ABB RAPID module: Module1.mod

MODULE Module1

! ## =========================================================================== ##
    ! MIT License
    ! Copyright (c) 2021 Roman Parak
    ! Permission is hereby granted, free of charge, to any person obtaining a copy
    ! of this software and associated documentation files (the "Software"), to deal
    ! in the Software without restriction, including without limitation the rights
    ! to use, copy, modify, merge, publish, distribute, sublicense, and/or sell
    ! copies of the Software, and to permit persons to whom the Software is
    ! furnished to do so, subject to the following conditions:
    ! The above copyright notice and this permission notice shall be included in all
    ! copies or substantial portions of the Software.
    ! THE SOFTWARE IS PROVIDED "AS IS", WITHOUT WARRANTY OF ANY KIND, EXPRESS OR
    ! IMPLIED, INCLUDING BUT NOT LIMITED TO THE WARRANTIES OF MERCHANTABILITY,
    ! FITNESS FOR A PARTICULAR PURPOSE AND NONINFRINGEMENT. IN NO EVENT SHALL THE
    ! AUTHORS OR COPYRIGHT HOLDERS BE LIABLE FOR ANY CLAIM, DAMAGES OR OTHER
    ! LIABILITY, WHETHER IN AN ACTION OF CONTRACT, TORT OR OTHERWISE, ARISING FROM,
    ! OUT OF OR IN CONNECTION WITH THE SOFTWARE OR THE USE OR OTHER DEALINGS IN THE
    ! SOFTWARE.
    ! ## =========================================================================== ##
    ! Author   : Roman Parak
    ! Email    : Roman.Parak@outlook.com
    ! Github   : https://github.com/rparak
    ! File Name: T_ROB1/Module1.mod
    ! ## =========================================================================== ##

    ! ############### EGM Initialization Parameters ############### !
    ! Identifier for the EGM correction.
     VAR robtarget starting_position;

    ! ################################## Externally Guided motion (EGM) - Main Cycle ################################## !
    PROC main()
        starting_position := CRobT(\Tool:=Tooldata_7\wobj:=wobj0);
        MoveJ RelTool (starting_position, 327, 6, -563 \Rx:=-9.8, \Ry:=17.7, \Rz:=0), v400, z1, Tooldata_7;
        MoveJ RelTool (starting_position, 326, 8, -564 \Rx:=-9.9, \Ry:=17.4, \Rz:=0), v400, z1, Tooldata_7;
        MoveJ RelTool (starting_position, 325, 10, -565 \Rx:=-9.9, \Ry:=17.1, \Rz:=0), v400, z1, Tooldata_7;
        MoveJ RelTool (starting_position, 324, 12, -566 \Rx:=-9.9, \Ry:=17.1, \Rz:=0), v400, z1, Tooldata_7;
        MoveJ RelTool (starting_position, 323, 14, -567 \Rx:=-9.9, \Ry:=16.8, \Rz:=0), v400, z1, Tooldata_7;
        MoveJ RelTool (starting_position, 321, 16, -568 \Rx:=-9.9, \Ry:=16.5, \Rz:=0), v400, z1, Tooldata_7;
        MoveJ RelTool (starting_position, 320, 20, -569 \Rx:=-10, \Ry:=16.2, \Rz:=0), v400, z1, Tooldata_7;
        MoveJ RelTool (starting_position, 318, 22, -570 \Rx:=-10, \Ry:=15.9, \Rz:=0), v400, z1, Tooldata_7;
        MoveJ RelTool (starting_position, 317, 26, -571 \Rx:=-10, \Ry:=15.6, \Rz:=0), v400, z1, Tooldata_7;
        MoveJ RelTool (starting_position, 315, 28, -572 \Rx:=-10, \Ry:=15.6, \Rz:=0), v400, z1, Tooldata_7;
        MoveJ RelTool (starting_position, 313, 32, -573 \Rx:=-10, \Ry:=15.3, \Rz:=0), v400, z1, Tooldata_7;
        MoveJ RelTool (starting_position, 311, 34, -574 \Rx:=-10, \Ry:=15, \Rz:=0), v400, z1, Tooldata_7;
        MoveJ RelTool (starting_position, 309, 38, -576 \Rx:=-10, \Ry:=14.7, \Rz:=0), v400, z1, Tooldata_7;
        MoveJ RelTool (starting_position, 307, 42, -577 \Rx:=-10, \Ry:=14.4, \Rz:=0), v400, z1, Tooldata_7;
        MoveJ RelTool (starting_position, 305, 44, -578 \Rx:=-9.9, \Ry:=14.1, \Rz:=0), v400, z1, Tooldata_7;
        MoveJ RelTool (starting_position, 302, 48, -580 \Rx:=-9.9, \Ry:=13.8, \Rz:=0), v400, z1, Tooldata_7;
        MoveJ RelTool (starting_position, 300, 52, -581 \Rx:=-9.8, \Ry:=13.5, \Rz:=0), v400, z1, Tooldata_7;
        MoveJ RelTool (starting_position, 298, 54, -583 \Rx:=-9.8, \Ry:=13.2, \Rz:=0), v400, z1, Tooldata_7;
        MoveJ RelTool (starting_position, 296, 58, -584 \Rx:=-9.7, \Ry:=12.9, \Rz:=0), v400, z1, Tooldata_7;
        MoveJ RelTool (starting_position, 293, 62, -586 \Rx:=-9.5, \Ry:=12.6, \Rz:=0), v400, z1, Tooldata_7;
        MoveJ RelTool (starting_position, 291, 64, -587 \Rx:=-9.4, \Ry:=12.3, \Rz:=0), v400, z1, Tooldata_7;
        MoveJ RelTool (starting_position, 288, 68, -589 \Rx:=-9.3, \Ry:=12, \Rz:=0), v400, z1, Tooldata_7;
        MoveJ RelTool (starting_position, 285, 72, -590 \Rx:=-9.2, \Ry:=11.7, \Rz:=0), v400, z1, Tooldata_7;
        MoveJ RelTool (starting_position, 283, 74, -592 \Rx:=-9.2, \Ry:=11.1, \Rz:=0), v400, z1, Tooldata_7;
        MoveJ RelTool (starting_position, 280, 78, -594 \Rx:=-9.1, \Ry:=10.8, \Rz:=0), v400, z1, Tooldata_7;
        MoveJ RelTool (starting_position, 277, 82, -595 \Rx:=-8.9, \Ry:=10.5, \Rz:=0), v400, z1, Tooldata_7;
        MoveJ RelTool (starting_position, 274, 84, -597 \Rx:=-8.8, \Ry:=10.2, \Rz:=0), v400, z1, Tooldata_7;
        MoveJ RelTool (starting_position, 270, 88, -598 \Rx:=-8.7, \Ry:=9.6, \Rz:=0), v400, z1, Tooldata_7;
        MoveJ RelTool (starting_position, 267, 92, -600 \Rx:=-8.6, \Ry:=9, \Rz:=0), v400, z1, Tooldata_7;
        MoveJ RelTool (starting_position, 263, 94, -601 \Rx:=-8.5, \Ry:=8.7, \Rz:=0), v400, z1, Tooldata_7;
        MoveJ RelTool (starting_position, 260, 98, -603 \Rx:=-8.4, \Ry:=8.1, \Rz:=0), v400, z1, Tooldata_7;
        MoveJ RelTool (starting_position, 256, 102, -604 \Rx:=-8.2, \Ry:=7.5, \Rz:=0), v400, z1, Tooldata_7;
        MoveJ RelTool (starting_position, 253, 104, -605 \Rx:=-8.1, \Ry:=6.9, \Rz:=0), v400, z1, Tooldata_7;
        MoveJ RelTool (starting_position, 249, 108, -606 \Rx:=-7.9, \Ry:=6.6, \Rz:=0), v400, z1, Tooldata_7;
        MoveJ RelTool (starting_position, 245, 112, -607 \Rx:=-7.6, \Ry:=6, \Rz:=0), v400, z1, Tooldata_7;
        MoveJ RelTool (starting_position, 242, 114, -608 \Rx:=-7.4, \Ry:=5.7, \Rz:=0), v400, z1, Tooldata_7;
        MoveJ RelTool (starting_position, 238, 118, -609 \Rx:=-7.1, \Ry:=5.1, \Rz:=0), v400, z1, Tooldata_7;
        MoveJ RelTool (starting_position, 234, 122, -609 \Rx:=-6.8, \Ry:=4.5, \Rz:=0), v400, z1, Tooldata_7;
        MoveJ RelTool (starting_position, 231, 124, -610 \Rx:=-6.6, \Ry:=4.2, \Rz:=0), v400, z1, Tooldata_7;
        MoveJ RelTool (starting_position, 227, 128, -610 \Rx:=-6.4, \Ry:=3.6, \Rz:=0), v400, z1, Tooldata_7;
        MoveJ RelTool (starting_position, 224, 130, -611 \Rx:=-6.1, \Ry:=3.3, \Rz:=0), v400, z1, Tooldata_7;
        MoveJ RelTool (starting_position, 220, 134, -611 \Rx:=-6, \Ry:=2.7, \Rz:=0), v400, z1, Tooldata_7;
        MoveJ RelTool (starting_position, 217, 136, -611 \Rx:=-5.9, \Ry:=2.1, \Rz:=0), v400, z1, Tooldata_7;
        MoveJ RelTool (starting_position, 213, 140, -611 \Rx:=-5.9, \Ry:=1.5, \Rz:=0), v400, z1, Tooldata_7;
        MoveJ RelTool (starting_position, 210, 142, -611 \Rx:=-5.9, \Ry:=1.2, \Rz:=0), v400, z1, Tooldata_7;
        MoveJ RelTool (starting_position, 207, 146, -611 \Rx:=-5.9, \Ry:=0.9, \Rz:=0), v400, z1, Tooldata_7;
        MoveJ RelTool (starting_position, 203, 148, -611 \Rx:=-6, \Ry:=0.3, \Rz:=0), v400, z1, Tooldata_7;
        MoveJ RelTool (starting_position, 200, 152, -610 \Rx:=-6.2, \Ry:=0, \Rz:=0), v400, z1, Tooldata_7;
        MoveJ RelTool (starting_position, 198, 156, -610 \Rx:=-6.4, \Ry:=-0.3, \Rz:=0), v400, z1, Tooldata_7;
        MoveJ RelTool (starting_position, 195, 158, -610 \Rx:=-6.6, \Ry:=-0.9, \Rz:=0), v400, z1, Tooldata_7;
        MoveJ RelTool (starting_position, 192, 162, -609 \Rx:=-6.8, \Ry:=-1.2, \Rz:=0), v400, z1, Tooldata_7;
        MoveJ RelTool (starting_position, 190, 164, -609 \Rx:=-7.1, \Ry:=-1.5, \Rz:=0), v400, z1, Tooldata_7;
        MoveJ RelTool (starting_position, 188, 168, -608 \Rx:=-7.5, \Ry:=-1.8, \Rz:=0), v400, z1, Tooldata_7;
        MoveJ RelTool (starting_position, 186, 170, -608 \Rx:=-7.8, \Ry:=-2.1, \Rz:=0), v400, z1, Tooldata_7;
        MoveJ RelTool (starting_position, 184, 174, -607 \Rx:=-8.2, \Ry:=-2.4, \Rz:=0), v400, z1, Tooldata_7;
        MoveJ RelTool (starting_position, 182, 176, -607 \Rx:=-8.7, \Ry:=-2.7, \Rz:=0), v400, z1, Tooldata_7;
        MoveJ RelTool (starting_position, 180, 180, -607 \Rx:=-9.1, \Ry:=-2.7, \Rz:=0), v400, z1, Tooldata_7;
        MoveJ RelTool (starting_position, 179, 182, -606 \Rx:=-9.4, \Ry:=-3, \Rz:=0), v400, z1, Tooldata_7;
        MoveJ RelTool (starting_position, 178, 186, -605 \Rx:=-9.8, \Ry:=-3, \Rz:=0), v400, z1, Tooldata_7;
        MoveJ RelTool (starting_position, 177, 188, -605 \Rx:=-10.2, \Ry:=-3.3, \Rz:=0), v400, z1, Tooldata_7;
        MoveJ RelTool (starting_position, 176, 192, -604 \Rx:=-10.6, \Ry:=-3.3, \Rz:=0), v400, z1, Tooldata_7;
        MoveJ RelTool (starting_position, 175, 194, -604 \Rx:=-11, \Ry:=-3.3, \Rz:=0), v400, z1, Tooldata_7;
        MoveJ RelTool (starting_position, 174, 198, -603 \Rx:=-11.3, \Ry:=-3.6, \Rz:=0), v400, z1, Tooldata_7;
        MoveJ RelTool (starting_position, 173, 200, -603 \Rx:=-11.7, \Ry:=-3.6, \Rz:=0), v400, z1, Tooldata_7;
        MoveJ RelTool (starting_position, 173, 202, -602 \Rx:=-12.1, \Ry:=-3.6, \Rz:=0), v400, z1, Tooldata_7;
        MoveJ RelTool (starting_position, 172, 206, -601 \Rx:=-12.4, \Ry:=-3.9, \Rz:=0), v400, z1, Tooldata_7;
        MoveJ RelTool (starting_position, 172, 208, -601 \Rx:=-12.7, \Ry:=-3.9, \Rz:=0), v400, z1, Tooldata_7;
        MoveJ RelTool (starting_position, 172, 212, -600 \Rx:=-12.9, \Ry:=-3.9, \Rz:=0), v400, z1, Tooldata_7;
        MoveJ RelTool (starting_position, 172, 214, -599 \Rx:=-13, \Ry:=-3.9, \Rz:=0), v400, z1, Tooldata_7;
        MoveJ RelTool (starting_position, 172, 218, -599 \Rx:=-13.1, \Ry:=-3.9, \Rz:=0), v400, z1, Tooldata_7;
        MoveJ RelTool (starting_position, 172, 220, -598 \Rx:=-13.1, \Ry:=-3.9, \Rz:=0), v400, z1, Tooldata_7;
        MoveJ RelTool (starting_position, 172, 222, -597 \Rx:=-13, \Ry:=-3.6, \Rz:=0), v400, z1, Tooldata_7;
        MoveJ RelTool (starting_position, 173, 226, -597 \Rx:=-12.9, \Ry:=-3.6, \Rz:=0), v400, z1, Tooldata_7;
        MoveJ RelTool (starting_position, 173, 228, -596 \Rx:=-12.5, \Ry:=-3.6, \Rz:=0), v400, z1, Tooldata_7;
        MoveJ RelTool (starting_position, 173, 230, -595 \Rx:=-12.2, \Ry:=-3.6, \Rz:=0), v400, z1, Tooldata_7;
        MoveJ RelTool (starting_position, 174, 234, -595 \Rx:=-11.8, \Ry:=-3.6, \Rz:=0), v400, z1, Tooldata_7;
        MoveJ RelTool (starting_position, 174, 236, -594 \Rx:=-11.3, \Ry:=-3.3, \Rz:=0), v400, z1, Tooldata_7;
        MoveJ RelTool (starting_position, 175, 238, -594 \Rx:=-10.7, \Ry:=-3.3, \Rz:=0), v400, z1, Tooldata_7;
        MoveJ RelTool (starting_position, 175, 242, -593 \Rx:=-10, \Ry:=-3.3, \Rz:=0), v400, z1, Tooldata_7;
        MoveJ RelTool (starting_position, 175, 244, -593 \Rx:=-9.2, \Ry:=-3.3, \Rz:=0), v400, z1, Tooldata_7;
        MoveJ RelTool (starting_position, 176, 246, -592 \Rx:=-8.4, \Ry:=-3.3, \Rz:=0), v400, z1, Tooldata_7;
        MoveJ RelTool (starting_position, 176, 248, -592 \Rx:=-7.6, \Ry:=-3, \Rz:=0), v400, z1, Tooldata_7;
        MoveJ RelTool (starting_position, 176, 252, -591 \Rx:=-6.7, \Ry:=-3, \Rz:=0), v400, z1, Tooldata_7;
        MoveJ RelTool (starting_position, 177, 254, -591 \Rx:=-5.8, \Ry:=-3, \Rz:=0), v400, z1, Tooldata_7;
        MoveJ RelTool (starting_position, 177, 258, -591 \Rx:=-5, \Ry:=-3, \Rz:=0), v400, z1, Tooldata_7;
        MoveJ RelTool (starting_position, 177, 260, -591 \Rx:=-4.2, \Ry:=-3, \Rz:=0), v400, z1, Tooldata_7;
        MoveJ RelTool (starting_position, 176, 262, -590 \Rx:=-3.5, \Ry:=-3, \Rz:=0), v400, z1, Tooldata_7;
        MoveJ RelTool (starting_position, 176, 266, -590 \Rx:=-2.8, \Ry:=-3, \Rz:=0), v400, z1, Tooldata_7;
        MoveJ RelTool (starting_position, 176, 268, -590 \Rx:=-2.2, \Ry:=-3, \Rz:=0), v400, z1, Tooldata_7;
        MoveJ RelTool (starting_position, 175, 270, -590 \Rx:=-1.5, \Ry:=-3.3, \Rz:=0), v400, z1, Tooldata_7;
        MoveJ RelTool (starting_position, 174, 274, -590 \Rx:=-1, \Ry:=-3.3, \Rz:=0), v400, z1, Tooldata_7;
        MoveJ RelTool (starting_position, 173, 276, -590 \Rx:=-0.5, \Ry:=-3.3, \Rz:=0), v400, z1, Tooldata_7;
        MoveJ RelTool (starting_position, 172, 278, -590 \Rx:=-0.1, \Ry:=-3.6, \Rz:=0), v400, z1, Tooldata_7;
        MoveJ RelTool (starting_position, 170, 280, -590 \Rx:=0.2, \Ry:=-3.6, \Rz:=0), v400, z1, Tooldata_7;
        MoveJ RelTool (starting_position, 168, 282, -590 \Rx:=0.5, \Ry:=-3.9, \Rz:=0), v400, z1, Tooldata_7;
        MoveJ RelTool (starting_position, 166, 284, -590 \Rx:=0.6, \Ry:=-4.2, \Rz:=0), v400, z1, Tooldata_7;
        MoveJ RelTool (starting_position, 164, 286, -590 \Rx:=0.6, \Ry:=-4.5, \Rz:=0), v400, z1, Tooldata_7;
        MoveJ RelTool (starting_position, 161, 288, -590 \Rx:=0.6, \Ry:=-4.8, \Rz:=0), v400, z1, Tooldata_7;
        MoveJ RelTool (starting_position, 159, 292, -590 \Rx:=0.6, \Ry:=-5.4, \Rz:=0), v400, z1, Tooldata_7;
        MoveJ RelTool (starting_position, 155, 294, -590 \Rx:=0.6, \Ry:=-5.7, \Rz:=0), v400, z1, Tooldata_7;
        MoveJ RelTool (starting_position, 152, 296, -589 \Rx:=0.5, \Ry:=-6.3, \Rz:=0), v400, z1, Tooldata_7;
        MoveJ RelTool (starting_position, 149, 298, -589 \Rx:=0.4, \Ry:=-6.6, \Rz:=0), v400, z1, Tooldata_7;
        MoveJ RelTool (starting_position, 145, 300, -589 \Rx:=0.4, \Ry:=-7.2, \Rz:=0), v400, z1, Tooldata_7;
        MoveJ RelTool (starting_position, 141, 302, -588 \Rx:=0.3, \Ry:=-7.8, \Rz:=0), v400, z1, Tooldata_7;
        MoveJ RelTool (starting_position, 137, 304, -588 \Rx:=0.3, \Ry:=-8.4, \Rz:=0), v400, z1, Tooldata_7;
        MoveJ RelTool (starting_position, 133, 306, -587 \Rx:=0.4, \Ry:=-9, \Rz:=0), v400, z1, Tooldata_7;
        MoveJ RelTool (starting_position, 129, 308, -586 \Rx:=0.4, \Ry:=-9.6, \Rz:=0), v400, z1, Tooldata_7;
        MoveJ RelTool (starting_position, 125, 310, -586 \Rx:=0.5, \Ry:=-10.2, \Rz:=0), v400, z1, Tooldata_7;
        MoveJ RelTool (starting_position, 120, 314, -585 \Rx:=0.6, \Ry:=-10.5, \Rz:=0), v400, z1, Tooldata_7;
        MoveJ RelTool (starting_position, 116, 316, -583 \Rx:=0.9, \Ry:=-11.1, \Rz:=0), v400, z1, Tooldata_7;
        MoveJ RelTool (starting_position, 111, 318, -582 \Rx:=1.2, \Ry:=-11.7, \Rz:=0), v400, z1, Tooldata_7;
        MoveJ RelTool (starting_position, 107, 318, -581 \Rx:=1.5, \Ry:=-12.3, \Rz:=0), v400, z1, Tooldata_7;
        MoveJ RelTool (starting_position, 102, 320, -579 \Rx:=1.9, \Ry:=-12.9, \Rz:=0), v400, z1, Tooldata_7;
        MoveJ RelTool (starting_position, 97, 322, -577 \Rx:=2.4, \Ry:=-13.8, \Rz:=0), v400, z1, Tooldata_7;
        MoveJ RelTool (starting_position, 92, 324, -575 \Rx:=2.8, \Ry:=-14.7, \Rz:=0), v400, z1, Tooldata_7;
        MoveJ RelTool (starting_position, 88, 326, -573 \Rx:=3.2, \Ry:=-15.3, \Rz:=0), v400, z1, Tooldata_7;
        MoveJ RelTool (starting_position, 83, 328, -571 \Rx:=3.7, \Ry:=-15.9, \Rz:=0), v400, z1, Tooldata_7;
        MoveJ RelTool (starting_position, 79, 330, -569 \Rx:=4.2, \Ry:=-16.5, \Rz:=0), v400, z1, Tooldata_7;
        MoveJ RelTool (starting_position, 74, 332, -566 \Rx:=4.7, \Ry:=-17.1, \Rz:=0), v400, z1, Tooldata_7;
        MoveJ RelTool (starting_position, 70, 334, -564 \Rx:=5.2, \Ry:=-17.7, \Rz:=0), v400, z1, Tooldata_7;
        MoveJ RelTool (starting_position, 66, 336, -561 \Rx:=5.6, \Ry:=-18, \Rz:=0), v400, z1, Tooldata_7;
        MoveJ RelTool (starting_position, 62, 338, -558 \Rx:=6.2, \Ry:=-18.6, \Rz:=0), v400, z1, Tooldata_7;
        MoveJ RelTool (starting_position, 59, 340, -555 \Rx:=6.7, \Ry:=-19.2, \Rz:=0), v400, z1, Tooldata_7;
        MoveJ RelTool (starting_position, 55, 342, -553 \Rx:=7.2, \Ry:=-19.5, \Rz:=0), v400, z1, Tooldata_7;
        MoveJ RelTool (starting_position, 52, 344, -550 \Rx:=7.6, \Ry:=-20.1, \Rz:=0), v400, z1, Tooldata_7;
        MoveJ RelTool (starting_position, 49, 344, -546 \Rx:=8.1, \Ry:=-20.4, \Rz:=0), v400, z1, Tooldata_7;
        MoveJ RelTool (starting_position, 46, 346, -543 \Rx:=8.6, \Ry:=-21, \Rz:=0), v400, z1, Tooldata_7;
        MoveJ RelTool (starting_position, 44, 348, -540 \Rx:=9, \Ry:=-21.3, \Rz:=0), v400, z1, Tooldata_7;
        MoveJ RelTool (starting_position, 41, 350, -537 \Rx:=9.4, \Ry:=-21.3, \Rz:=0), v400, z1, Tooldata_7;
        MoveJ RelTool (starting_position, 39, 352, -534 \Rx:=9.8, \Ry:=-21.9, \Rz:=0), v400, z1, Tooldata_7;
        MoveJ RelTool (starting_position, 37, 354, -530 \Rx:=10.2, \Ry:=-22.2, \Rz:=0), v400, z1, Tooldata_7;
        MoveJ RelTool (starting_position, 36, 356, -527 \Rx:=10.6, \Ry:=-22.2, \Rz:=0), v400, z1, Tooldata_7;
        MoveJ RelTool (starting_position, 34, 358, -524 \Rx:=10.9, \Ry:=-22.5, \Rz:=0), v400, z1, Tooldata_7;
        MoveJ RelTool (starting_position, 33, 358, -521 \Rx:=11.2, \Ry:=-22.5, \Rz:=0), v400, z1, Tooldata_7;
        MoveJ RelTool (starting_position, 32, 360, -517 \Rx:=11.5, \Ry:=-22.8, \Rz:=0), v400, z1, Tooldata_7;
        MoveJ RelTool (starting_position, 32, 360, -514 \Rx:=11.9, \Ry:=-22.8, \Rz:=0), v400, z1, Tooldata_7;
        MoveJ RelTool (starting_position, 31, 362, -511 \Rx:=12.2, \Ry:=-22.8, \Rz:=0), v400, z1, Tooldata_7;
        MoveJ RelTool (starting_position, 31, 362, -507 \Rx:=12.5, \Ry:=-22.8, \Rz:=0), v400, z1, Tooldata_7;
        MoveJ RelTool (starting_position, 31, 364, -504 \Rx:=12.8, \Ry:=-22.8, \Rz:=0), v400, z1, Tooldata_7;
        MoveJ RelTool (starting_position, 31, 366, -501 \Rx:=13, \Ry:=-22.8, \Rz:=0), v400, z1, Tooldata_7;
        MoveJ RelTool (starting_position, 31, 366, -498 \Rx:=13.3, \Ry:=-22.8, \Rz:=0), v400, z1, Tooldata_7;
        MoveJ RelTool (starting_position, 31, 368, -495 \Rx:=13.5, \Ry:=-22.8, \Rz:=0), v400, z1, Tooldata_7;
        MoveJ RelTool (starting_position, 31, 370, -492 \Rx:=13.7, \Ry:=-22.8, \Rz:=0), v400, z1, Tooldata_7;
        MoveJ RelTool (starting_position, 32, 372, -488 \Rx:=13.9, \Ry:=-22.8, \Rz:=0), v400, z1, Tooldata_7;
        MoveJ RelTool (starting_position, 32, 374, -485 \Rx:=14.1, \Ry:=-22.5, \Rz:=0), v400, z1, Tooldata_7;
        MoveJ RelTool (starting_position, 33, 376, -482 \Rx:=14.2, \Ry:=-22.5, \Rz:=0), v400, z1, Tooldata_7;
        MoveJ RelTool (starting_position, 34, 378, -479 \Rx:=14.3, \Ry:=-22.2, \Rz:=0), v400, z1, Tooldata_7;
        MoveJ RelTool (starting_position, 35, 378, -476 \Rx:=14.3, \Ry:=-22.2, \Rz:=0), v400, z1, Tooldata_7;
        MoveJ RelTool (starting_position, 36, 380, -473 \Rx:=14.3, \Ry:=-22.2, \Rz:=0), v400, z1, Tooldata_7;
        MoveJ RelTool (starting_position, 37, 380, -470 \Rx:=14.2, \Ry:=-21.9, \Rz:=0), v400, z1, Tooldata_7;
        MoveJ RelTool (starting_position, 38, 380, -467 \Rx:=14.1, \Ry:=-21.6, \Rz:=0), v400, z1, Tooldata_7;
        MoveJ RelTool (starting_position, 39, 380, -465 \Rx:=13.8, \Ry:=-21.6, \Rz:=0), v400, z1, Tooldata_7;
        MoveJ RelTool (starting_position, 40, 380, -462 \Rx:=13.5, \Ry:=-21.3, \Rz:=0), v400, z1, Tooldata_7;
        MoveJ RelTool (starting_position, 41, 380, -459 \Rx:=13.1, \Ry:=-21.3, \Rz:=0), v400, z1, Tooldata_7;
        MoveJ RelTool (starting_position, 43, 380, -456 \Rx:=12.6, \Ry:=-21, \Rz:=0), v400, z1, Tooldata_7;
        MoveJ RelTool (starting_position, 44, 380, -453 \Rx:=12.1, \Ry:=-21, \Rz:=0), v400, z1, Tooldata_7;
        MoveJ RelTool (starting_position, 45, 382, -451 \Rx:=11.5, \Ry:=-20.7, \Rz:=0), v400, z1, Tooldata_7;
        MoveJ RelTool (starting_position, 46, 382, -448 \Rx:=10.8, \Ry:=-20.7, \Rz:=0), v400, z1, Tooldata_7;
        MoveJ RelTool (starting_position, 47, 384, -445 \Rx:=10.1, \Ry:=-20.4, \Rz:=0), v400, z1, Tooldata_7;
        MoveJ RelTool (starting_position, 48, 386, -442 \Rx:=9.2, \Ry:=-20.4, \Rz:=0), v400, z1, Tooldata_7;
        MoveJ RelTool (starting_position, 49, 386, -440 \Rx:=8.3, \Ry:=-20.1, \Rz:=0), v400, z1, Tooldata_7;
        MoveJ RelTool (starting_position, 50, 388, -437 \Rx:=7.3, \Ry:=-20.1, \Rz:=0), v400, z1, Tooldata_7;
        MoveJ RelTool (starting_position, 51, 390, -434 \Rx:=6.3, \Ry:=-20.1, \Rz:=0), v400, z1, Tooldata_7;
        MoveJ RelTool (starting_position, 52, 392, -432 \Rx:=5.2, \Ry:=-19.8, \Rz:=0), v400, z1, Tooldata_7;
        MoveJ RelTool (starting_position, 52, 394, -429 \Rx:=4.2, \Ry:=-19.8, \Rz:=0), v400, z1, Tooldata_7;
        MoveJ RelTool (starting_position, 53, 396, -427 \Rx:=3.1, \Ry:=-19.5, \Rz:=0), v400, z1, Tooldata_7;
        MoveJ RelTool (starting_position, 54, 398, -424 \Rx:=2.1, \Ry:=-19.5, \Rz:=0), v400, z1, Tooldata_7;
        MoveJ RelTool (starting_position, 55, 398, -422 \Rx:=1.1, \Ry:=-19.5, \Rz:=0), v400, z1, Tooldata_7;
        MoveJ RelTool (starting_position, 55, 400, -419 \Rx:=0.1, \Ry:=-19.2, \Rz:=0), v400, z1, Tooldata_7;
        MoveJ RelTool (starting_position, 56, 400, -417 \Rx:=-0.9, \Ry:=-19.2, \Rz:=0), v400, z1, Tooldata_7;
        MoveJ RelTool (starting_position, 57, 400, -415 \Rx:=-1.8, \Ry:=-19.2, \Rz:=0), v400, z1, Tooldata_7;
        MoveJ RelTool (starting_position, 57, 400, -413 \Rx:=-2.6, \Ry:=-19.2, \Rz:=0), v400, z1, Tooldata_7;
        MoveJ RelTool (starting_position, 58, 400, -410 \Rx:=-3.3, \Ry:=-19.2, \Rz:=0), v400, z1, Tooldata_7;
        MoveJ RelTool (starting_position, 58, 400, -408 \Rx:=-3.8, \Ry:=-18.9, \Rz:=0), v400, z1, Tooldata_7;
        MoveJ RelTool (starting_position, 59, 400, -406 \Rx:=-4.1, \Ry:=-18.9, \Rz:=0), v400, z1, Tooldata_7;
        MoveJ RelTool (starting_position, 59, 400, -404 \Rx:=-4.4, \Ry:=-18.9, \Rz:=0), v400, z1, Tooldata_7;
        MoveJ RelTool (starting_position, 60, 400, -402 \Rx:=-4.6, \Ry:=-18.9, \Rz:=0), v400, z1, Tooldata_7;
        MoveJ RelTool (starting_position, 60, 400, -400 \Rx:=-4.6, \Ry:=-18.6, \Rz:=0), v400, z1, Tooldata_7;
        MoveJ RelTool (starting_position, 61, 400, -398 \Rx:=-4.5, \Ry:=-18.6, \Rz:=0), v400, z1, Tooldata_7;
        MoveJ RelTool (starting_position, 61, 400, -395 \Rx:=-4.2, \Ry:=-18.6, \Rz:=0), v400, z1, Tooldata_7;
        MoveJ RelTool (starting_position, 62, 400, -393 \Rx:=-3.9, \Ry:=-18.6, \Rz:=0), v400, z1, Tooldata_7;
        MoveJ RelTool (starting_position, 62, 400, -391 \Rx:=-3.4, \Ry:=-18.6, \Rz:=0), v400, z1, Tooldata_7;
        MoveJ RelTool (starting_position, 63, 400, -389 \Rx:=-2.7, \Ry:=-18.6, \Rz:=0), v400, z1, Tooldata_7;
        MoveJ RelTool (starting_position, 63, 400, -386 \Rx:=-2, \Ry:=-18.3, \Rz:=0), v400, z1, Tooldata_7;
        MoveJ RelTool (starting_position, 64, 400, -384 \Rx:=-1.3, \Ry:=-18.3, \Rz:=0), v400, z1, Tooldata_7;
        MoveJ RelTool (starting_position, 65, 400, -381 \Rx:=-0.5, \Ry:=-18.3, \Rz:=0), v400, z1, Tooldata_7;
        MoveJ RelTool (starting_position, 66, 400, -379 \Rx:=0.3, \Ry:=-18, \Rz:=0), v400, z1, Tooldata_7;
        MoveJ RelTool (starting_position, 67, 400, -376 \Rx:=1.2, \Ry:=-18, \Rz:=0), v400, z1, Tooldata_7;
        MoveJ RelTool (starting_position, 68, 400, -374 \Rx:=2, \Ry:=-17.7, \Rz:=0), v400, z1, Tooldata_7;
        MoveJ RelTool (starting_position, 70, 400, -371 \Rx:=2.9, \Ry:=-17.7, \Rz:=0), v400, z1, Tooldata_7;
        MoveJ RelTool (starting_position, 71, 400, -368 \Rx:=3.7, \Ry:=-17.4, \Rz:=0), v400, z1, Tooldata_7;
        MoveJ RelTool (starting_position, 73, 400, -366 \Rx:=4.5, \Ry:=-17.1, \Rz:=0), v400, z1, Tooldata_7;
        MoveJ RelTool (starting_position, 75, 400, -363 \Rx:=5.4, \Ry:=-17.1, \Rz:=0), v400, z1, Tooldata_7;
        MoveJ RelTool (starting_position, 77, 400, -360 \Rx:=6.2, \Ry:=-16.8, \Rz:=0), v400, z1, Tooldata_7;
        MoveJ RelTool (starting_position, 79, 400, -357 \Rx:=6.9, \Ry:=-16.2, \Rz:=0), v400, z1, Tooldata_7;
        MoveJ RelTool (starting_position, 81, 400, -355 \Rx:=7.6, \Ry:=-15.9, \Rz:=0), v400, z1, Tooldata_7;
        MoveJ RelTool (starting_position, 84, 400, -352 \Rx:=8.2, \Ry:=-15.6, \Rz:=0), v400, z1, Tooldata_7;
        MoveJ RelTool (starting_position, 86, 400, -349 \Rx:=8.8, \Ry:=-15.3, \Rz:=0), v400, z1, Tooldata_7;
        MoveJ RelTool (starting_position, 89, 400, -347 \Rx:=9.3, \Ry:=-15, \Rz:=0), v400, z1, Tooldata_7;
        MoveJ RelTool (starting_position, 92, 400, -345 \Rx:=9.7, \Ry:=-14.7, \Rz:=0), v400, z1, Tooldata_7;
        MoveJ RelTool (starting_position, 95, 400, -342 \Rx:=10.1, \Ry:=-14.1, \Rz:=0), v400, z1, Tooldata_7;
        MoveJ RelTool (starting_position, 98, 400, -340 \Rx:=10.4, \Ry:=-13.8, \Rz:=0), v400, z1, Tooldata_7;
        MoveJ RelTool (starting_position, 101, 400, -338 \Rx:=10.5, \Ry:=-13.2, \Rz:=0), v400, z1, Tooldata_7;
        MoveJ RelTool (starting_position, 104, 400, -336 \Rx:=10.6, \Ry:=-12.9, \Rz:=0), v400, z1, Tooldata_7;
        MoveJ RelTool (starting_position, 107, 400, -335 \Rx:=10.7, \Ry:=-12.3, \Rz:=0), v400, z1, Tooldata_7;
        MoveJ RelTool (starting_position, 110, 400, -333 \Rx:=10.6, \Ry:=-12, \Rz:=0), v400, z1, Tooldata_7;
        MoveJ RelTool (starting_position, 112, 400, -332 \Rx:=10.5, \Ry:=-11.7, \Rz:=0), v400, z1, Tooldata_7;
        MoveJ RelTool (starting_position, 115, 400, -331 \Rx:=10.3, \Ry:=-11.1, \Rz:=0), v400, z1, Tooldata_7;
        MoveJ RelTool (starting_position, 118, 400, -329 \Rx:=10.1, \Ry:=-10.8, \Rz:=0), v400, z1, Tooldata_7;
        MoveJ RelTool (starting_position, 120, 400, -329 \Rx:=9.9, \Ry:=-10.5, \Rz:=0), v400, z1, Tooldata_7;
        MoveJ RelTool (starting_position, 122, 398, -328 \Rx:=9.6, \Ry:=-10.2, \Rz:=0), v400, z1, Tooldata_7;
        MoveJ RelTool (starting_position, 124, 398, -327 \Rx:=9.3, \Ry:=-9.9, \Rz:=0), v400, z1, Tooldata_7;
        MoveJ RelTool (starting_position, 125, 396, -327 \Rx:=8.9, \Ry:=-9.6, \Rz:=0), v400, z1, Tooldata_7;
        MoveJ RelTool (starting_position, 127, 394, -326 \Rx:=8.6, \Ry:=-9.6, \Rz:=0), v400, z1, Tooldata_7;
        MoveJ RelTool (starting_position, 128, 394, -326 \Rx:=8.3, \Ry:=-9.3, \Rz:=0), v400, z1, Tooldata_7;
        MoveJ RelTool (starting_position, 128, 392, -325 \Rx:=8, \Ry:=-9.3, \Rz:=0), v400, z1, Tooldata_7;
        MoveJ RelTool (starting_position, 129, 390, -325 \Rx:=7.7, \Ry:=-9.3, \Rz:=0), v400, z1, Tooldata_7;
        MoveJ RelTool (starting_position, 129, 388, -325 \Rx:=7.5, \Ry:=-9.3, \Rz:=0), v400, z1, Tooldata_7;
        MoveJ RelTool (starting_position, 129, 386, -324 \Rx:=7.4, \Ry:=-9.3, \Rz:=0), v400, z1, Tooldata_7;
        MoveJ RelTool (starting_position, 128, 384, -324 \Rx:=7.3, \Ry:=-9.3, \Rz:=0), v400, z1, Tooldata_7;
        MoveJ RelTool (starting_position, 128, 382, -324 \Rx:=7.3, \Ry:=-9.3, \Rz:=0), v400, z1, Tooldata_7;
        MoveJ RelTool (starting_position, 127, 382, -323 \Rx:=7.3, \Ry:=-9.6, \Rz:=0), v400, z1, Tooldata_7;
        MoveJ RelTool (starting_position, 125, 380, -323 \Rx:=7.3, \Ry:=-9.6, \Rz:=0), v400, z1, Tooldata_7;
        MoveJ RelTool (starting_position, 124, 380, -322 \Rx:=7.4, \Ry:=-9.9, \Rz:=0), v400, z1, Tooldata_7;
        MoveJ RelTool (starting_position, 122, 380, -321 \Rx:=7.6, \Ry:=-10.2, \Rz:=0), v400, z1, Tooldata_7;
        MoveJ RelTool (starting_position, 120, 380, -321 \Rx:=7.8, \Ry:=-10.5, \Rz:=0), v400, z1, Tooldata_7;
        MoveJ RelTool (starting_position, 118, 380, -320 \Rx:=8.1, \Ry:=-10.8, \Rz:=0), v400, z1, Tooldata_7;
        MoveJ RelTool (starting_position, 115, 380, -319 \Rx:=8.3, \Ry:=-11.1, \Rz:=0), v400, z1, Tooldata_7;
        MoveJ RelTool (starting_position, 113, 380, -317 \Rx:=8.6, \Ry:=-11.7, \Rz:=0), v400, z1, Tooldata_7;
        MoveJ RelTool (starting_position, 110, 380, -316 \Rx:=8.8, \Ry:=-12, \Rz:=0), v400, z1, Tooldata_7;
        MoveJ RelTool (starting_position, 108, 378, -315 \Rx:=9.1, \Ry:=-12.6, \Rz:=0), v400, z1, Tooldata_7;
        MoveJ RelTool (starting_position, 105, 378, -313 \Rx:=9.4, \Ry:=-12.9, \Rz:=0), v400, z1, Tooldata_7;
        MoveJ RelTool (starting_position, 102, 376, -311 \Rx:=9.7, \Ry:=-13.2, \Rz:=0), v400, z1, Tooldata_7;
        MoveJ RelTool (starting_position, 100, 374, -309 \Rx:=9.9, \Ry:=-13.5, \Rz:=0), v400, z1, Tooldata_7;
        MoveJ RelTool (starting_position, 98, 374, -307 \Rx:=10.1, \Ry:=-13.8, \Rz:=0), v400, z1, Tooldata_7;
        MoveJ RelTool (starting_position, 95, 372, -305 \Rx:=10.4, \Ry:=-14.1, \Rz:=0), v400, z1, Tooldata_7;
        MoveJ RelTool (starting_position, 93, 370, -303 \Rx:=10.6, \Ry:=-14.4, \Rz:=0), v400, z1, Tooldata_7;
        MoveJ RelTool (starting_position, 91, 368, -301 \Rx:=10.7, \Ry:=-14.7, \Rz:=0), v400, z1, Tooldata_7;
        MoveJ RelTool (starting_position, 89, 366, -298 \Rx:=10.9, \Ry:=-15, \Rz:=0), v400, z1, Tooldata_7;
        MoveJ RelTool (starting_position, 88, 364, -296 \Rx:=11, \Ry:=-15.3, \Rz:=0), v400, z1, Tooldata_7;
        MoveJ RelTool (starting_position, 86, 362, -293 \Rx:=11, \Ry:=-15.6, \Rz:=0), v400, z1, Tooldata_7;
        MoveJ RelTool (starting_position, 85, 362, -291 \Rx:=11, \Ry:=-15.6, \Rz:=0), v400, z1, Tooldata_7;
        MoveJ RelTool (starting_position, 84, 360, -288 \Rx:=10.9, \Ry:=-15.9, \Rz:=0), v400, z1, Tooldata_7;
        MoveJ RelTool (starting_position, 83, 360, -286 \Rx:=10.9, \Ry:=-15.9, \Rz:=0), v400, z1, Tooldata_7;
        MoveJ RelTool (starting_position, 83, 358, -283 \Rx:=10.8, \Ry:=-16.2, \Rz:=0), v400, z1, Tooldata_7;
        MoveJ RelTool (starting_position, 82, 358, -281 \Rx:=10.7, \Ry:=-15.9, \Rz:=0), v400, z1, Tooldata_7;
        MoveJ RelTool (starting_position, 82, 356, -278 \Rx:=10.6, \Ry:=-15.9, \Rz:=0), v400, z1, Tooldata_7;
        MoveJ RelTool (starting_position, 82, 354, -275 \Rx:=10.5, \Ry:=-15.9, \Rz:=0), v400, z1, Tooldata_7;
        MoveJ RelTool (starting_position, 83, 354, -273 \Rx:=10.3, \Ry:=-15.9, \Rz:=0), v400, z1, Tooldata_7;
        MoveJ RelTool (starting_position, 83, 352, -270 \Rx:=10.2, \Ry:=-15.9, \Rz:=0), v400, z1, Tooldata_7;
        MoveJ RelTool (starting_position, 84, 350, -268 \Rx:=10.1, \Ry:=-15.6, \Rz:=0), v400, z1, Tooldata_7;
        MoveJ RelTool (starting_position, 85, 348, -266 \Rx:=9.9, \Ry:=-15.6, \Rz:=0), v400, z1, Tooldata_7;
        MoveJ RelTool (starting_position, 86, 346, -263 \Rx:=9.8, \Ry:=-15.3, \Rz:=0), v400, z1, Tooldata_7;
        MoveJ RelTool (starting_position, 88, 344, -261 \Rx:=9.7, \Ry:=-15.3, \Rz:=0), v400, z1, Tooldata_7;
        MoveJ RelTool (starting_position, 89, 342, -259 \Rx:=9.6, \Ry:=-15, \Rz:=0), v400, z1, Tooldata_7;
        MoveJ RelTool (starting_position, 90, 340, -256 \Rx:=9.5, \Ry:=-14.7, \Rz:=0), v400, z1, Tooldata_7;
        MoveJ RelTool (starting_position, 92, 338, -254 \Rx:=9.4, \Ry:=-14.4, \Rz:=0), v400, z1, Tooldata_7;
        MoveJ RelTool (starting_position, 94, 336, -252 \Rx:=9.3, \Ry:=-14.4, \Rz:=0), v400, z1, Tooldata_7;
        MoveJ RelTool (starting_position, 95, 336, -250 \Rx:=9.2, \Ry:=-14.1, \Rz:=0), v400, z1, Tooldata_7;
        MoveJ RelTool (starting_position, 97, 334, -248 \Rx:=9.2, \Ry:=-13.8, \Rz:=0), v400, z1, Tooldata_7;
        MoveJ RelTool (starting_position, 99, 332, -246 \Rx:=9.1, \Ry:=-13.5, \Rz:=0), v400, z1, Tooldata_7;
        MoveJ RelTool (starting_position, 100, 330, -245 \Rx:=9, \Ry:=-13.2, \Rz:=0), v400, z1, Tooldata_7;
        MoveJ RelTool (starting_position, 102, 326, -243 \Rx:=8.9, \Ry:=-12.9, \Rz:=0), v400, z1, Tooldata_7;
        MoveJ RelTool (starting_position, 103, 324, -241 \Rx:=8.8, \Ry:=-12.9, \Rz:=0), v400, z1, Tooldata_7;
        MoveJ RelTool (starting_position, 105, 322, -240 \Rx:=8.6, \Ry:=-12.6, \Rz:=0), v400, z1, Tooldata_7;
        MoveJ RelTool (starting_position, 106, 322, -238 \Rx:=8.5, \Ry:=-12.3, \Rz:=0), v400, z1, Tooldata_7;
        MoveJ RelTool (starting_position, 107, 320, -237 \Rx:=8.4, \Ry:=-12.3, \Rz:=0), v400, z1, Tooldata_7;
        MoveJ RelTool (starting_position, 107, 318, -236 \Rx:=8.2, \Ry:=-12.3, \Rz:=0), v400, z1, Tooldata_7;
        MoveJ RelTool (starting_position, 108, 316, -234 \Rx:=8, \Ry:=-12, \Rz:=0), v400, z1, Tooldata_7;
        MoveJ RelTool (starting_position, 108, 314, -233 \Rx:=7.8, \Ry:=-12, \Rz:=0), v400, z1, Tooldata_7;
        MoveJ RelTool (starting_position, 108, 312, -232 \Rx:=7.5, \Ry:=-12, \Rz:=0), v400, z1, Tooldata_7;
        MoveJ RelTool (starting_position, 107, 308, -232 \Rx:=7.2, \Ry:=-12, \Rz:=0), v400, z1, Tooldata_7;
        MoveJ RelTool (starting_position, 106, 306, -231 \Rx:=6.9, \Ry:=-12, \Rz:=0), v400, z1, Tooldata_7;
        MoveJ RelTool (starting_position, 105, 304, -230 \Rx:=6.6, \Ry:=-12.3, \Rz:=0), v400, z1, Tooldata_7;
        MoveJ RelTool (starting_position, 103, 302, -230 \Rx:=6.4, \Ry:=-12.6, \Rz:=0), v400, z1, Tooldata_7;
        MoveJ RelTool (starting_position, 101, 300, -229 \Rx:=6.1, \Ry:=-12.9, \Rz:=0), v400, z1, Tooldata_7;
        MoveJ RelTool (starting_position, 98, 298, -228 \Rx:=5.9, \Ry:=-13.2, \Rz:=0), v400, z1, Tooldata_7;
        MoveJ RelTool (starting_position, 95, 296, -228 \Rx:=5.7, \Ry:=-13.8, \Rz:=0), v400, z1, Tooldata_7;
        MoveJ RelTool (starting_position, 91, 294, -227 \Rx:=5.6, \Ry:=-14.1, \Rz:=0), v400, z1, Tooldata_7;
        MoveJ RelTool (starting_position, 87, 292, -227 \Rx:=5.4, \Ry:=-14.7, \Rz:=0), v400, z1, Tooldata_7;
        MoveJ RelTool (starting_position, 83, 288, -226 \Rx:=5.3, \Ry:=-15.3, \Rz:=0), v400, z1, Tooldata_7;
        MoveJ RelTool (starting_position, 79, 286, -225 \Rx:=5.3, \Ry:=-16.2, \Rz:=0), v400, z1, Tooldata_7;
        MoveJ RelTool (starting_position, 74, 284, -224 \Rx:=5.3, \Ry:=-16.8, \Rz:=0), v400, z1, Tooldata_7;
        MoveJ RelTool (starting_position, 68, 282, -223 \Rx:=5.3, \Ry:=-17.4, \Rz:=0), v400, z1, Tooldata_7;
        MoveJ RelTool (starting_position, 63, 280, -222 \Rx:=5.3, \Ry:=-18, \Rz:=0), v400, z1, Tooldata_7;
        MoveJ RelTool (starting_position, 57, 278, -220 \Rx:=5.4, \Ry:=-18.9, \Rz:=0), v400, z1, Tooldata_7;
        MoveJ RelTool (starting_position, 51, 276, -219 \Rx:=5.4, \Ry:=-19.5, \Rz:=0), v400, z1, Tooldata_7;
        MoveJ RelTool (starting_position, 45, 274, -217 \Rx:=5.5, \Ry:=-20.7, \Rz:=0), v400, z1, Tooldata_7;
        MoveJ RelTool (starting_position, 39, 270, -214 \Rx:=5.6, \Ry:=-21.6, \Rz:=0), v400, z1, Tooldata_7;
        MoveJ RelTool (starting_position, 32, 268, -212 \Rx:=5.6, \Ry:=-22.5, \Rz:=0), v400, z1, Tooldata_7;
        MoveJ RelTool (starting_position, 26, 266, -209 \Rx:=5.7, \Ry:=-23.4, \Rz:=0), v400, z1, Tooldata_7;
        MoveJ RelTool (starting_position, 19, 262, -206 \Rx:=5.8, \Ry:=-24.3, \Rz:=0), v400, z1, Tooldata_7;
        MoveJ RelTool (starting_position, 13, 260, -202 \Rx:=6, \Ry:=-25.2, \Rz:=0), v400, z1, Tooldata_7;
        MoveJ RelTool (starting_position, 6, 258, -199 \Rx:=6, \Ry:=-26.1, \Rz:=0), v400, z1, Tooldata_7;
        MoveJ RelTool (starting_position, 0, 254, -195 \Rx:=6, \Ry:=-27, \Rz:=0), v400, z1, Tooldata_7;
        MoveJ RelTool (starting_position, -6, 252, -191 \Rx:=6, \Ry:=-27.9, \Rz:=0), v400, z1, Tooldata_7;
        MoveJ RelTool (starting_position, -12, 250, -186 \Rx:=5.9, \Ry:=-28.8, \Rz:=0), v400, z1, Tooldata_7;
        MoveJ RelTool (starting_position, -18, 246, -182 \Rx:=5.8, \Ry:=-29.7, \Rz:=0), v400, z1, Tooldata_7;
        MoveJ RelTool (starting_position, -23, 244, -177 \Rx:=5.7, \Ry:=-30.3, \Rz:=0), v400, z1, Tooldata_7;
        MoveJ RelTool (starting_position, -28, 242, -172 \Rx:=5.6, \Ry:=-31.2, \Rz:=0), v400, z1, Tooldata_7;
        MoveJ RelTool (starting_position, -32, 238, -167 \Rx:=5.4, \Ry:=-31.5, \Rz:=0), v400, z1, Tooldata_7;
        MoveJ RelTool (starting_position, -36, 236, -162 \Rx:=5.2, \Ry:=-32.1, \Rz:=0), v400, z1, Tooldata_7;
        MoveJ RelTool (starting_position, -40, 234, -157 \Rx:=5, \Ry:=-32.7, \Rz:=0), v400, z1, Tooldata_7;
        MoveJ RelTool (starting_position, -43, 232, -152 \Rx:=4.7, \Ry:=-33, \Rz:=0), v400, z1, Tooldata_7;
        MoveJ RelTool (starting_position, -46, 228, -146 \Rx:=4.4, \Ry:=-33.3, \Rz:=0), v400, z1, Tooldata_7;
        MoveJ RelTool (starting_position, -48, 226, -141 \Rx:=4, \Ry:=-33.6, \Rz:=0), v400, z1, Tooldata_7;
        MoveJ RelTool (starting_position, -50, 222, -136 \Rx:=3.7, \Ry:=-33.9, \Rz:=0), v400, z1, Tooldata_7;
        MoveJ RelTool (starting_position, -51, 220, -131 \Rx:=3.4, \Ry:=-34.2, \Rz:=0), v400, z1, Tooldata_7;
        MoveJ RelTool (starting_position, -52, 218, -126 \Rx:=3.1, \Ry:=-34.2, \Rz:=0), v400, z1, Tooldata_7;
        MoveJ RelTool (starting_position, -53, 214, -121 \Rx:=2.8, \Ry:=-34.2, \Rz:=0), v400, z1, Tooldata_7;
        MoveJ RelTool (starting_position, -54, 212, -116 \Rx:=2.5, \Ry:=-34.2, \Rz:=0), v400, z1, Tooldata_7;
        MoveJ RelTool (starting_position, -54, 208, -111 \Rx:=2.1, \Ry:=-34.2, \Rz:=0), v400, z1, Tooldata_7;
        MoveJ RelTool (starting_position, -54, 206, -107 \Rx:=1.8, \Ry:=-34.2, \Rz:=0), v400, z1, Tooldata_7;
        MoveJ RelTool (starting_position, -53, 202, -102 \Rx:=1.6, \Ry:=-34.2, \Rz:=0), v400, z1, Tooldata_7;
        MoveJ RelTool (starting_position, -53, 200, -98 \Rx:=1.3, \Ry:=-34.2, \Rz:=0), v400, z1, Tooldata_7;
        MoveJ RelTool (starting_position, -52, 198, -93 \Rx:=1.1, \Ry:=-34.2, \Rz:=0), v400, z1, Tooldata_7;
        MoveJ RelTool (starting_position, -51, 194, -89 \Rx:=0.8, \Ry:=-33.9, \Rz:=0), v400, z1, Tooldata_7;
        MoveJ RelTool (starting_position, -50, 192, -85 \Rx:=0.7, \Ry:=-33.6, \Rz:=0), v400, z1, Tooldata_7;
        MoveJ RelTool (starting_position, -48, 188, -80 \Rx:=0.6, \Ry:=-33.3, \Rz:=0), v400, z1, Tooldata_7;
        MoveJ RelTool (starting_position, -47, 186, -76 \Rx:=0.6, \Ry:=-33, \Rz:=0), v400, z1, Tooldata_7;
        MoveJ RelTool (starting_position, -46, 182, -72 \Rx:=0.7, \Ry:=-33, \Rz:=0), v400, z1, Tooldata_7;
        MoveJ RelTool (starting_position, -44, 180, -68 \Rx:=0.8, \Ry:=-32.7, \Rz:=0), v400, z1, Tooldata_7;
        MoveJ RelTool (starting_position, -42, 178, -64 \Rx:=1, \Ry:=-32.7, \Rz:=0), v400, z1, Tooldata_7;
        MoveJ RelTool (starting_position, -40, 174, -60 \Rx:=1.3, \Ry:=-32.4, \Rz:=0), v400, z1, Tooldata_7;
        MoveJ RelTool (starting_position, -38, 172, -56 \Rx:=1.6, \Ry:=-32.1, \Rz:=0), v400, z1, Tooldata_7;
        MoveJ RelTool (starting_position, -36, 168, -52 \Rx:=2, \Ry:=-31.8, \Rz:=0), v400, z1, Tooldata_7;
        MoveJ RelTool (starting_position, -34, 164, -47 \Rx:=2.5, \Ry:=-31.5, \Rz:=0), v400, z1, Tooldata_7;
        MoveJ RelTool (starting_position, -31, 162, -43 \Rx:=3, \Ry:=-31.2, \Rz:=0), v400, z1, Tooldata_7;
        MoveJ RelTool (starting_position, -29, 158, -39 \Rx:=3.5, \Ry:=-30.9, \Rz:=0), v400, z1, Tooldata_7;
        MoveJ RelTool (starting_position, -26, 156, -35 \Rx:=4.1, \Ry:=-30.3, \Rz:=0), v400, z1, Tooldata_7;
        MoveJ RelTool (starting_position, -23, 152, -31 \Rx:=4.8, \Ry:=-30, \Rz:=0), v400, z1, Tooldata_7;
        MoveJ RelTool (starting_position, -20, 150, -26 \Rx:=5.4, \Ry:=-29.7, \Rz:=0), v400, z1, Tooldata_7;
        MoveJ RelTool (starting_position, -17, 146, -22 \Rx:=6.1, \Ry:=-29.1, \Rz:=0), v400, z1, Tooldata_7;
        MoveJ RelTool (starting_position, -14, 144, -18 \Rx:=6.8, \Ry:=-28.8, \Rz:=0), v400, z1, Tooldata_7;
        MoveJ RelTool (starting_position, -11, 140, -14 \Rx:=7.5, \Ry:=-28.2, \Rz:=0), v400, z1, Tooldata_7;
        MoveJ RelTool (starting_position, -8, 138, -10 \Rx:=8.1, \Ry:=-27.9, \Rz:=0), v400, z1, Tooldata_7;
        MoveJ RelTool (starting_position, -5, 134, -6 \Rx:=8.8, \Ry:=-27.3, \Rz:=0), v400, z1, Tooldata_7;
        MoveJ RelTool (starting_position, -2, 132, -2 \Rx:=9.3, \Ry:=-27, \Rz:=0), v400, z1, Tooldata_7;
        MoveJ RelTool (starting_position, 1, 128, 2 \Rx:=9.9, \Ry:=-26.4, \Rz:=0), v400, z1, Tooldata_7;
        MoveJ RelTool (starting_position, 4, 124, 6 \Rx:=10.4, \Ry:=-26.1, \Rz:=0), v400, z1, Tooldata_7;
        MoveJ RelTool (starting_position, 7, 122, 10 \Rx:=10.9, \Ry:=-25.8, \Rz:=0), v400, z1, Tooldata_7;
        MoveJ RelTool (starting_position, 10, 118, 13 \Rx:=11.3, \Ry:=-25.5, \Rz:=0), v400, z1, Tooldata_7;
        MoveJ RelTool (starting_position, 13, 116, 17 \Rx:=11.7, \Ry:=-25.2, \Rz:=0), v400, z1, Tooldata_7;
        MoveJ RelTool (starting_position, 16, 112, 20 \Rx:=12, \Ry:=-24.6, \Rz:=0), v400, z1, Tooldata_7;
        MoveJ RelTool (starting_position, 19, 108, 23 \Rx:=12.3, \Ry:=-24.3, \Rz:=0), v400, z1, Tooldata_7;
        MoveJ RelTool (starting_position, 21, 106, 26 \Rx:=12.5, \Ry:=-24, \Rz:=0), v400, z1, Tooldata_7;
        MoveJ RelTool (starting_position, 24, 102, 29 \Rx:=12.7, \Ry:=-23.4, \Rz:=0), v400, z1, Tooldata_7;
        MoveJ RelTool (starting_position, 27, 98, 32 \Rx:=12.8, \Ry:=-23.1, \Rz:=0), v400, z1, Tooldata_7;
        MoveJ RelTool (starting_position, 29, 96, 35 \Rx:=12.9, \Ry:=-22.8, \Rz:=0), v400, z1, Tooldata_7;
        MoveJ RelTool (starting_position, 32, 92, 37 \Rx:=13, \Ry:=-22.2, \Rz:=0), v400, z1, Tooldata_7;
        MoveJ RelTool (starting_position, 34, 88, 40 \Rx:=13, \Ry:=-22.2, \Rz:=0), v400, z1, Tooldata_7;
        MoveJ RelTool (starting_position, 36, 86, 42 \Rx:=13, \Ry:=-21.9, \Rz:=0), v400, z1, Tooldata_7;
        MoveJ RelTool (starting_position, 39, 82, 45 \Rx:=13, \Ry:=-21.6, \Rz:=0), v400, z1, Tooldata_7;
        MoveJ RelTool (starting_position, 41, 78, 48 \Rx:=12.9, \Ry:=-21.3, \Rz:=0), v400, z1, Tooldata_7;
        MoveJ RelTool (starting_position, 43, 76, 50 \Rx:=12.9, \Ry:=-21, \Rz:=0), v400, z1, Tooldata_7;
        MoveJ RelTool (starting_position, 45, 72, 53 \Rx:=12.8, \Ry:=-20.7, \Rz:=0), v400, z1, Tooldata_7;
        MoveJ RelTool (starting_position, 47, 68, 55 \Rx:=12.8, \Ry:=-20.4, \Rz:=0), v400, z1, Tooldata_7;
        MoveJ RelTool (starting_position, 49, 66, 58 \Rx:=12.7, \Ry:=-20.1, \Rz:=0), v400, z1, Tooldata_7;
        MoveJ RelTool (starting_position, 50, 62, 60 \Rx:=12.6, \Ry:=-20.1, \Rz:=0), v400, z1, Tooldata_7;
        MoveJ RelTool (starting_position, 52, 58, 63 \Rx:=12.4, \Ry:=-19.8, \Rz:=0), v400, z1, Tooldata_7;
        MoveJ RelTool (starting_position, 54, 56, 65 \Rx:=12.3, \Ry:=-19.5, \Rz:=0), v400, z1, Tooldata_7;
        MoveJ RelTool (starting_position, 56, 52, 68 \Rx:=12.2, \Ry:=-19.2, \Rz:=0), v400, z1, Tooldata_7;
        MoveJ RelTool (starting_position, 57, 48, 70 \Rx:=12, \Ry:=-19.2, \Rz:=0), v400, z1, Tooldata_7;
        MoveJ RelTool (starting_position, 59, 46, 73 \Rx:=11.9, \Ry:=-18.9, \Rz:=0), v400, z1, Tooldata_7;
        MoveJ RelTool (starting_position, 61, 42, 75 \Rx:=11.7, \Ry:=-18.9, \Rz:=0), v400, z1, Tooldata_7;
        MoveJ RelTool (starting_position, 63, 38, 78 \Rx:=11.6, \Ry:=-18.6, \Rz:=0), v400, z1, Tooldata_7;
        MoveJ RelTool (starting_position, 65, 36, 80 \Rx:=11.4, \Ry:=-18.3, \Rz:=0), v400, z1, Tooldata_7;
        MoveJ RelTool (starting_position, 67, 32, 83 \Rx:=11.3, \Ry:=-18, \Rz:=0), v400, z1, Tooldata_7;
        MoveJ RelTool (starting_position, 69, 28, 86 \Rx:=11.1, \Ry:=-17.4, \Rz:=0), v400, z1, Tooldata_7;
        MoveJ RelTool (starting_position, 71, 26, 88 \Rx:=11, \Ry:=-17.4, \Rz:=0), v400, z1, Tooldata_7;
        MoveJ RelTool (starting_position, 73, 22, 91 \Rx:=10.8, \Ry:=-17.1, \Rz:=0), v400, z1, Tooldata_7;
        MoveJ RelTool (starting_position, 76, 18, 93 \Rx:=10.7, \Ry:=-16.8, \Rz:=0), v400, z1, Tooldata_7;
        MoveJ RelTool (starting_position, 79, 16, 96 \Rx:=10.6, \Ry:=-16.5, \Rz:=0), v400, z1, Tooldata_7;
        MoveJ RelTool (starting_position, 81, 12, 98 \Rx:=10.4, \Ry:=-15.9, \Rz:=0), v400, z1, Tooldata_7;
        MoveJ RelTool (starting_position, 84, 8, 101 \Rx:=10.3, \Ry:=-15.6, \Rz:=0), v400, z1, Tooldata_7;
        MoveJ RelTool (starting_position, 87, 6, 103 \Rx:=10.2, \Ry:=-15.3, \Rz:=0), v400, z1, Tooldata_7;
        MoveJ RelTool (starting_position, 90, 2, 106 \Rx:=10.1, \Ry:=-14.7, \Rz:=0), v400, z1, Tooldata_7;
        MoveJ RelTool (starting_position, 94, -2, 108 \Rx:=10.1, \Ry:=-14.4, \Rz:=0), v400, z1, Tooldata_7;
        MoveJ RelTool (starting_position, 97, -4, 110 \Rx:=10, \Ry:=-13.8, \Rz:=0), v400, z1, Tooldata_7;
        MoveJ RelTool (starting_position, 100, -8, 113 \Rx:=10, \Ry:=-13.5, \Rz:=0), v400, z1, Tooldata_7;
        MoveJ RelTool (starting_position, 104, -12, 115 \Rx:=10, \Ry:=-12.9, \Rz:=0), v400, z1, Tooldata_7;
        MoveJ RelTool (starting_position, 107, -14, 117 \Rx:=10, \Ry:=-12.6, \Rz:=0), v400, z1, Tooldata_7;
        MoveJ RelTool (starting_position, 111, -18, 119 \Rx:=10, \Ry:=-12, \Rz:=0), v400, z1, Tooldata_7;
        MoveJ RelTool (starting_position, 115, -22, 121 \Rx:=10, \Ry:=-11.4, \Rz:=0), v400, z1, Tooldata_7;
        MoveJ RelTool (starting_position, 119, -24, 123 \Rx:=10.1, \Ry:=-10.8, \Rz:=0), v400, z1, Tooldata_7;
        MoveJ RelTool (starting_position, 123, -28, 124 \Rx:=10.2, \Ry:=-10.2, \Rz:=0), v400, z1, Tooldata_7;
        MoveJ RelTool (starting_position, 127, -30, 126 \Rx:=10.2, \Ry:=-9.9, \Rz:=0), v400, z1, Tooldata_7;
        MoveJ RelTool (starting_position, 131, -34, 127 \Rx:=10.3, \Ry:=-9.3, \Rz:=0), v400, z1, Tooldata_7;
        MoveJ RelTool (starting_position, 135, -36, 129 \Rx:=10.4, \Ry:=-8.7, \Rz:=0), v400, z1, Tooldata_7;
        MoveJ RelTool (starting_position, 139, -40, 130 \Rx:=10.4, \Ry:=-8.1, \Rz:=0), v400, z1, Tooldata_7;
        MoveJ RelTool (starting_position, 143, -42, 131 \Rx:=10.4, \Ry:=-7.5, \Rz:=0), v400, z1, Tooldata_7;
        MoveJ RelTool (starting_position, 147, -46, 131 \Rx:=10.5, \Ry:=-6.9, \Rz:=0), v400, z1, Tooldata_7;
        MoveJ RelTool (starting_position, 150, -48, 132 \Rx:=10.5, \Ry:=-6.3, \Rz:=0), v400, z1, Tooldata_7;
        MoveJ RelTool (starting_position, 154, -52, 132 \Rx:=10.5, \Ry:=-6, \Rz:=0), v400, z1, Tooldata_7;
        MoveJ RelTool (starting_position, 157, -56, 133 \Rx:=10.6, \Ry:=-5.4, \Rz:=0), v400, z1, Tooldata_7;
        MoveJ RelTool (starting_position, 160, -58, 133 \Rx:=10.6, \Ry:=-4.8, \Rz:=0), v400, z1, Tooldata_7;
        MoveJ RelTool (starting_position, 163, -62, 133 \Rx:=10.6, \Ry:=-4.5, \Rz:=0), v400, z1, Tooldata_7;
        MoveJ RelTool (starting_position, 166, -64, 133 \Rx:=10.5, \Ry:=-4.5, \Rz:=0), v400, z1, Tooldata_7;
        MoveJ RelTool (starting_position, 168, -68, 133 \Rx:=10.4, \Ry:=-4.2, \Rz:=0), v400, z1, Tooldata_7;
        MoveJ RelTool (starting_position, 170, -72, 133 \Rx:=10.4, \Ry:=-3.9, \Rz:=0), v400, z1, Tooldata_7;
        MoveJ RelTool (starting_position, 172, -74, 133 \Rx:=10.4, \Ry:=-3.6, \Rz:=0), v400, z1, Tooldata_7;
        MoveJ RelTool (starting_position, 174, -78, 132 \Rx:=10.3, \Ry:=-3.3, \Rz:=0), v400, z1, Tooldata_7;
        MoveJ RelTool (starting_position, 175, -82, 132 \Rx:=10.1, \Ry:=-3, \Rz:=0), v400, z1, Tooldata_7;
        MoveJ RelTool (starting_position, 177, -84, 132 \Rx:=10, \Ry:=-2.7, \Rz:=0), v400, z1, Tooldata_7;
        MoveJ RelTool (starting_position, 178, -88, 131 \Rx:=9.8, \Ry:=-2.7, \Rz:=0), v400, z1, Tooldata_7;
        MoveJ RelTool (starting_position, 179, -92, 131 \Rx:=9.6, \Ry:=-2.4, \Rz:=0), v400, z1, Tooldata_7;
        MoveJ RelTool (starting_position, 179, -94, 131 \Rx:=9.4, \Ry:=-2.4, \Rz:=0), v400, z1, Tooldata_7;
        MoveJ RelTool (starting_position, 179, -98, 131 \Rx:=9.2, \Ry:=-2.4, \Rz:=0), v400, z1, Tooldata_7;
        MoveJ RelTool (starting_position, 179, -102, 131 \Rx:=9, \Ry:=-2.7, \Rz:=0), v400, z1, Tooldata_7;
        MoveJ RelTool (starting_position, 179, -104, 131 \Rx:=8.9, \Ry:=-2.7, \Rz:=0), v400, z1, Tooldata_7;
        MoveJ RelTool (starting_position, 179, -108, 131 \Rx:=8.7, \Ry:=-2.7, \Rz:=0), v400, z1, Tooldata_7;
        MoveJ RelTool (starting_position, 178, -112, 131 \Rx:=8.5, \Ry:=-2.7, \Rz:=0), v400, z1, Tooldata_7;
        MoveJ RelTool (starting_position, 177, -114, 131 \Rx:=8.3, \Ry:=-3, \Rz:=0), v400, z1, Tooldata_7;
        MoveJ RelTool (starting_position, 177, -118, 131 \Rx:=8.2, \Ry:=-3, \Rz:=0), v400, z1, Tooldata_7;
        MoveJ RelTool (starting_position, 176, -122, 131 \Rx:=8, \Ry:=-3.3, \Rz:=0), v400, z1, Tooldata_7;
        MoveJ RelTool (starting_position, 175, -124, 132 \Rx:=7.8, \Ry:=-3.3, \Rz:=0), v400, z1, Tooldata_7;
        MoveJ RelTool (starting_position, 174, -128, 132 \Rx:=7.7, \Ry:=-3.6, \Rz:=0), v400, z1, Tooldata_7;
        MoveJ RelTool (starting_position, 174, -130, 133 \Rx:=7.5, \Ry:=-3.6, \Rz:=0), v400, z1, Tooldata_7;
        MoveJ RelTool (starting_position, 173, -134, 133 \Rx:=7.2, \Ry:=-3.6, \Rz:=0), v400, z1, Tooldata_7;
        MoveJ RelTool (starting_position, 172, -136, 134 \Rx:=7, \Ry:=-3.9, \Rz:=0), v400, z1, Tooldata_7;
        MoveJ RelTool (starting_position, 172, -140, 134 \Rx:=6.8, \Ry:=-3.9, \Rz:=0), v400, z1, Tooldata_7;
        MoveJ RelTool (starting_position, 171, -142, 135 \Rx:=6.5, \Ry:=-3.9, \Rz:=0), v400, z1, Tooldata_7;
        MoveJ RelTool (starting_position, 171, -146, 136 \Rx:=6.3, \Ry:=-3.9, \Rz:=0), v400, z1, Tooldata_7;
        MoveJ RelTool (starting_position, 170, -148, 137 \Rx:=6, \Ry:=-3.9, \Rz:=0), v400, z1, Tooldata_7;
        MoveJ RelTool (starting_position, 170, -152, 137 \Rx:=5.8, \Ry:=-3.9, \Rz:=0), v400, z1, Tooldata_7;
        MoveJ RelTool (starting_position, 170, -156, 138 \Rx:=5.5, \Ry:=-4.2, \Rz:=0), v400, z1, Tooldata_7;
        MoveJ RelTool (starting_position, 170, -158, 139 \Rx:=5.3, \Ry:=-4.2, \Rz:=0), v400, z1, Tooldata_7;
        MoveJ RelTool (starting_position, 171, -162, 140 \Rx:=5, \Ry:=-4.2, \Rz:=0), v400, z1, Tooldata_7;
        MoveJ RelTool (starting_position, 171, -164, 141 \Rx:=4.7, \Ry:=-4.2, \Rz:=0), v400, z1, Tooldata_7;
        MoveJ RelTool (starting_position, 172, -168, 142 \Rx:=4.5, \Ry:=-4.2, \Rz:=0), v400, z1, Tooldata_7;
        MoveJ RelTool (starting_position, 173, -170, 143 \Rx:=4.2, \Ry:=-3.9, \Rz:=0), v400, z1, Tooldata_7;
        MoveJ RelTool (starting_position, 174, -174, 144 \Rx:=3.9, \Ry:=-3.6, \Rz:=0), v400, z1, Tooldata_7;
        MoveJ RelTool (starting_position, 175, -176, 145 \Rx:=3.7, \Ry:=-3.3, \Rz:=0), v400, z1, Tooldata_7;
        MoveJ RelTool (starting_position, 177, -180, 146 \Rx:=3.3, \Ry:=-3.3, \Rz:=0), v400, z1, Tooldata_7;
        MoveJ RelTool (starting_position, 179, -182, 147 \Rx:=2.9, \Ry:=-3, \Rz:=0), v400, z1, Tooldata_7;
        MoveJ RelTool (starting_position, 181, -186, 148 \Rx:=2.5, \Ry:=-2.7, \Rz:=0), v400, z1, Tooldata_7;
        MoveJ RelTool (starting_position, 184, -188, 149 \Rx:=2.1, \Ry:=-2.4, \Rz:=0), v400, z1, Tooldata_7;
        MoveJ RelTool (starting_position, 186, -192, 150 \Rx:=1.7, \Ry:=-2.1, \Rz:=0), v400, z1, Tooldata_7;
        MoveJ RelTool (starting_position, 189, -194, 151 \Rx:=1.4, \Ry:=-1.5, \Rz:=0), v400, z1, Tooldata_7;
        MoveJ RelTool (starting_position, 192, -198, 151 \Rx:=1.2, \Ry:=-1.2, \Rz:=0), v400, z1, Tooldata_7;
        MoveJ RelTool (starting_position, 195, -200, 152 \Rx:=0.9, \Ry:=-0.9, \Rz:=0), v400, z1, Tooldata_7;
        MoveJ RelTool (starting_position, 198, -202, 152 \Rx:=0.7, \Ry:=-0.3, \Rz:=0), v400, z1, Tooldata_7;
        MoveJ RelTool (starting_position, 201, -206, 152 \Rx:=0.5, \Ry:=0.3, \Rz:=0), v400, z1, Tooldata_7;
        MoveJ RelTool (starting_position, 205, -208, 153 \Rx:=0.3, \Ry:=0.6, \Rz:=0), v400, z1, Tooldata_7;
        MoveJ RelTool (starting_position, 208, -212, 153 \Rx:=0.1, \Ry:=1.2, \Rz:=0), v400, z1, Tooldata_7;
        MoveJ RelTool (starting_position, 212, -214, 153 \Rx:=0.1, \Ry:=1.5, \Rz:=0), v400, z1, Tooldata_7;
        MoveJ RelTool (starting_position, 215, -218, 152 \Rx:=0.2, \Ry:=2.1, \Rz:=0), v400, z1, Tooldata_7;
        MoveJ RelTool (starting_position, 218, -220, 152 \Rx:=0.3, \Ry:=2.7, \Rz:=0), v400, z1, Tooldata_7;
        MoveJ RelTool (starting_position, 222, -222, 151 \Rx:=0.5, \Ry:=3.3, \Rz:=0), v400, z1, Tooldata_7;
        MoveJ RelTool (starting_position, 225, -226, 150 \Rx:=0.7, \Ry:=3.6, \Rz:=0), v400, z1, Tooldata_7;
        MoveJ RelTool (starting_position, 228, -228, 149 \Rx:=1, \Ry:=3.9, \Rz:=0), v400, z1, Tooldata_7;
        MoveJ RelTool (starting_position, 231, -230, 148 \Rx:=1.3, \Ry:=4.2, \Rz:=0), v400, z1, Tooldata_7;
        MoveJ RelTool (starting_position, 233, -234, 147 \Rx:=1.7, \Ry:=4.8, \Rz:=0), v400, z1, Tooldata_7;
        MoveJ RelTool (starting_position, 235, -236, 146 \Rx:=2.1, \Ry:=5.1, \Rz:=0), v400, z1, Tooldata_7;
        MoveJ RelTool (starting_position, 237, -238, 144 \Rx:=2.6, \Ry:=5.4, \Rz:=0), v400, z1, Tooldata_7;
        MoveJ RelTool (starting_position, 239, -242, 143 \Rx:=3, \Ry:=5.7, \Rz:=0), v400, z1, Tooldata_7;
        MoveJ RelTool (starting_position, 240, -244, 141 \Rx:=3.5, \Ry:=5.7, \Rz:=0), v400, z1, Tooldata_7;
        MoveJ RelTool (starting_position, 241, -246, 139 \Rx:=4, \Ry:=6, \Rz:=0), v400, z1, Tooldata_7;
        MoveJ RelTool (starting_position, 242, -248, 138 \Rx:=4.5, \Ry:=6, \Rz:=0), v400, z1, Tooldata_7;
        MoveJ RelTool (starting_position, 243, -252, 136 \Rx:=5, \Ry:=6, \Rz:=0), v400, z1, Tooldata_7;
        MoveJ RelTool (starting_position, 243, -254, 134 \Rx:=5.5, \Ry:=6, \Rz:=0), v400, z1, Tooldata_7;
        MoveJ RelTool (starting_position, 242, -258, 132 \Rx:=6, \Ry:=6, \Rz:=0), v400, z1, Tooldata_7;
        MoveJ RelTool (starting_position, 242, -260, 131 \Rx:=6.5, \Ry:=6, \Rz:=0), v400, z1, Tooldata_7;
        MoveJ RelTool (starting_position, 241, -262, 129 \Rx:=6.9, \Ry:=6, \Rz:=0), v400, z1, Tooldata_7;
        MoveJ RelTool (starting_position, 240, -266, 127 \Rx:=7.3, \Ry:=5.7, \Rz:=0), v400, z1, Tooldata_7;
        MoveJ RelTool (starting_position, 239, -268, 126 \Rx:=7.7, \Ry:=5.4, \Rz:=0), v400, z1, Tooldata_7;
        MoveJ RelTool (starting_position, 237, -270, 124 \Rx:=8.1, \Ry:=5.1, \Rz:=0), v400, z1, Tooldata_7;
        MoveJ RelTool (starting_position, 235, -274, 123 \Rx:=8.6, \Ry:=5.1, \Rz:=0), v400, z1, Tooldata_7;
        MoveJ RelTool (starting_position, 233, -276, 122 \Rx:=9, \Ry:=4.5, \Rz:=0), v400, z1, Tooldata_7;
        MoveJ RelTool (starting_position, 231, -278, 121 \Rx:=9.3, \Ry:=4.2, \Rz:=0), v400, z1, Tooldata_7;
        MoveJ RelTool (starting_position, 228, -280, 120 \Rx:=9.7, \Ry:=3.9, \Rz:=0), v400, z1, Tooldata_7;
        MoveJ RelTool (starting_position, 226, -282, 119 \Rx:=10, \Ry:=3.6, \Rz:=0), v400, z1, Tooldata_7;
        MoveJ RelTool (starting_position, 223, -284, 119 \Rx:=10.3, \Ry:=3.3, \Rz:=0), v400, z1, Tooldata_7;
        MoveJ RelTool (starting_position, 221, -286, 118 \Rx:=10.6, \Ry:=2.7, \Rz:=0), v400, z1, Tooldata_7;
        MoveJ RelTool (starting_position, 218, -288, 118 \Rx:=10.8, \Ry:=2.4, \Rz:=0), v400, z1, Tooldata_7;
        MoveJ RelTool (starting_position, 216, -292, 118 \Rx:=11, \Ry:=2.1, \Rz:=0), v400, z1, Tooldata_7;
        MoveJ RelTool (starting_position, 214, -294, 118 \Rx:=11.3, \Ry:=1.8, \Rz:=0), v400, z1, Tooldata_7;
        MoveJ RelTool (starting_position, 211, -296, 118 \Rx:=11.5, \Ry:=1.5, \Rz:=0), v400, z1, Tooldata_7;
        MoveJ RelTool (starting_position, 209, -298, 118 \Rx:=11.7, \Ry:=0.9, \Rz:=0), v400, z1, Tooldata_7;
        MoveJ RelTool (starting_position, 207, -300, 119 \Rx:=11.9, \Ry:=0.9, \Rz:=0), v400, z1, Tooldata_7;
        MoveJ RelTool (starting_position, 205, -302, 119 \Rx:=12.1, \Ry:=0.6, \Rz:=0), v400, z1, Tooldata_7;
        MoveJ RelTool (starting_position, 204, -304, 120 \Rx:=12.3, \Ry:=0.3, \Rz:=0), v400, z1, Tooldata_7;
        MoveJ RelTool (starting_position, 202, -306, 121 \Rx:=12.5, \Ry:=-0, \Rz:=0), v400, z1, Tooldata_7;
        MoveJ RelTool (starting_position, 201, -308, 122 \Rx:=12.8, \Ry:=-0.3, \Rz:=0), v400, z1, Tooldata_7;
        MoveJ RelTool (starting_position, 200, -310, 124 \Rx:=13, \Ry:=-0.3, \Rz:=0), v400, z1, Tooldata_7;
        MoveJ RelTool (starting_position, 200, -314, 125 \Rx:=13.3, \Ry:=-0.3, \Rz:=0), v400, z1, Tooldata_7;
        MoveJ RelTool (starting_position, 200, -316, 127 \Rx:=13.6, \Ry:=-0.3, \Rz:=0), v400, z1, Tooldata_7;
        MoveJ RelTool (starting_position, 200, -318, 128 \Rx:=13.7, \Ry:=-0.3, \Rz:=0), v400, z1, Tooldata_7;
        MoveJ RelTool (starting_position, 200, -318, 130 \Rx:=13.9, \Ry:=-0, \Rz:=0), v400, z1, Tooldata_7;
        MoveJ RelTool (starting_position, 201, -320, 131 \Rx:=14.1, \Ry:=-0, \Rz:=0), v400, z1, Tooldata_7;
        MoveJ RelTool (starting_position, 202, -322, 133 \Rx:=14.2, \Ry:=-0, \Rz:=0), v400, z1, Tooldata_7;
        MoveJ RelTool (starting_position, 204, -324, 135 \Rx:=14.4, \Ry:=0, \Rz:=0), v400, z1, Tooldata_7;
        MoveJ RelTool (starting_position, 206, -326, 136 \Rx:=14.5, \Ry:=0.3, \Rz:=0), v400, z1, Tooldata_7;
        MoveJ RelTool (starting_position, 208, -328, 138 \Rx:=14.6, \Ry:=0.6, \Rz:=0), v400, z1, Tooldata_7;
        MoveJ RelTool (starting_position, 210, -330, 140 \Rx:=14.6, \Ry:=1.2, \Rz:=0), v400, z1, Tooldata_7;
        MoveJ RelTool (starting_position, 213, -332, 141 \Rx:=14.6, \Ry:=1.5, \Rz:=0), v400, z1, Tooldata_7;
        MoveJ RelTool (starting_position, 217, -334, 142 \Rx:=14.5, \Ry:=2.1, \Rz:=0), v400, z1, Tooldata_7;
        MoveJ RelTool (starting_position, 220, -336, 144 \Rx:=14.4, \Ry:=2.4, \Rz:=0), v400, z1, Tooldata_7;
        MoveJ RelTool (starting_position, 224, -338, 145 \Rx:=14.3, \Ry:=2.7, \Rz:=0), v400, z1, Tooldata_7;
        MoveJ RelTool (starting_position, 229, -340, 145 \Rx:=14.1, \Ry:=3.6, \Rz:=0), v400, z1, Tooldata_7;
        MoveJ RelTool (starting_position, 233, -342, 146 \Rx:=13.9, \Ry:=4.2, \Rz:=0), v400, z1, Tooldata_7;
        MoveJ RelTool (starting_position, 238, -344, 146 \Rx:=13.6, \Ry:=4.8, \Rz:=0), v400, z1, Tooldata_7;
        MoveJ RelTool (starting_position, 243, -344, 146 \Rx:=13.3, \Ry:=5.7, \Rz:=0), v400, z1, Tooldata_7;
        MoveJ RelTool (starting_position, 249, -346, 146 \Rx:=13, \Ry:=6.6, \Rz:=0), v400, z1, Tooldata_7;
        MoveJ RelTool (starting_position, 254, -348, 146 \Rx:=12.7, \Ry:=7.2, \Rz:=0), v400, z1, Tooldata_7;
        MoveJ RelTool (starting_position, 260, -350, 145 \Rx:=12.4, \Ry:=8.1, \Rz:=0), v400, z1, Tooldata_7;
        MoveJ RelTool (starting_position, 266, -352, 144 \Rx:=12.1, \Ry:=9, \Rz:=0), v400, z1, Tooldata_7;
        MoveJ RelTool (starting_position, 271, -354, 143 \Rx:=11.8, \Ry:=9.9, \Rz:=0), v400, z1, Tooldata_7;
        MoveJ RelTool (starting_position, 277, -356, 142 \Rx:=11.5, \Ry:=10.5, \Rz:=0), v400, z1, Tooldata_7;
        MoveJ RelTool (starting_position, 282, -358, 141 \Rx:=11.1, \Ry:=11.4, \Rz:=0), v400, z1, Tooldata_7;
        MoveJ RelTool (starting_position, 288, -358, 139 \Rx:=10.9, \Ry:=12, \Rz:=0), v400, z1, Tooldata_7;
        MoveJ RelTool (starting_position, 293, -360, 138 \Rx:=10.6, \Ry:=12.6, \Rz:=0), v400, z1, Tooldata_7;
        MoveJ RelTool (starting_position, 298, -360, 136 \Rx:=10.3, \Ry:=13.2, \Rz:=0), v400, z1, Tooldata_7;
        MoveJ RelTool (starting_position, 302, -362, 134 \Rx:=10.1, \Ry:=13.8, \Rz:=0), v400, z1, Tooldata_7;
        MoveJ RelTool (starting_position, 307, -362, 131 \Rx:=9.8, \Ry:=14.7, \Rz:=0), v400, z1, Tooldata_7;
        MoveJ RelTool (starting_position, 311, -364, 129 \Rx:=9.6, \Ry:=15.3, \Rz:=0), v400, z1, Tooldata_7;
        MoveJ RelTool (starting_position, 315, -366, 127 \Rx:=9.4, \Ry:=15.9, \Rz:=0), v400, z1, Tooldata_7;
        MoveJ RelTool (starting_position, 319, -366, 124 \Rx:=9.1, \Ry:=16.5, \Rz:=0), v400, z1, Tooldata_7;
        MoveJ RelTool (starting_position, 322, -368, 122 \Rx:=8.9, \Ry:=16.8, \Rz:=0), v400, z1, Tooldata_7;
        MoveJ RelTool (starting_position, 325, -370, 120 \Rx:=8.6, \Ry:=17.1, \Rz:=0), v400, z1, Tooldata_7;
        MoveJ RelTool (starting_position, 328, -372, 118 \Rx:=8.4, \Ry:=17.4, \Rz:=0), v400, z1, Tooldata_7;
        MoveJ RelTool (starting_position, 330, -374, 115 \Rx:=8.1, \Ry:=17.7, \Rz:=0), v400, z1, Tooldata_7;
        MoveJ RelTool (starting_position, 333, -376, 113 \Rx:=7.8, \Ry:=18, \Rz:=0), v400, z1, Tooldata_7;
        MoveJ RelTool (starting_position, 335, -378, 111 \Rx:=7.5, \Ry:=18.3, \Rz:=0), v400, z1, Tooldata_7;
        MoveJ RelTool (starting_position, 337, -378, 109 \Rx:=7.1, \Ry:=18.6, \Rz:=0), v400, z1, Tooldata_7;
        MoveJ RelTool (starting_position, 338, -380, 107 \Rx:=6.7, \Ry:=18.9, \Rz:=0), v400, z1, Tooldata_7;
        MoveJ RelTool (starting_position, 340, -380, 106 \Rx:=6.3, \Ry:=18.9, \Rz:=0), v400, z1, Tooldata_7;
        MoveJ RelTool (starting_position, 341, -380, 104 \Rx:=5.8, \Ry:=19.2, \Rz:=0), v400, z1, Tooldata_7;
        MoveJ RelTool (starting_position, 341, -380, 103 \Rx:=5.3, \Ry:=19.2, \Rz:=0), v400, z1, Tooldata_7;
        MoveJ RelTool (starting_position, 342, -380, 101 \Rx:=4.8, \Ry:=19.5, \Rz:=0), v400, z1, Tooldata_7;
        MoveJ RelTool (starting_position, 342, -380, 100 \Rx:=4.2, \Ry:=19.5, \Rz:=0), v400, z1, Tooldata_7;
        MoveJ RelTool (starting_position, 342, -380, 98 \Rx:=3.6, \Ry:=19.5, \Rz:=0), v400, z1, Tooldata_7;
        MoveJ RelTool (starting_position, 342, -380, 97 \Rx:=2.9, \Ry:=19.5, \Rz:=0), v400, z1, Tooldata_7;
        MoveJ RelTool (starting_position, 341, -382, 95 \Rx:=2.1, \Ry:=19.2, \Rz:=0), v400, z1, Tooldata_7;
        MoveJ RelTool (starting_position, 340, -382, 94 \Rx:=1.3, \Ry:=19.2, \Rz:=0), v400, z1, Tooldata_7;
        MoveJ RelTool (starting_position, 339, -384, 92 \Rx:=0.5, \Ry:=18.9, \Rz:=0), v400, z1, Tooldata_7;
        MoveJ RelTool (starting_position, 337, -386, 90 \Rx:=-0.3, \Ry:=18.6, \Rz:=0), v400, z1, Tooldata_7;
        MoveJ RelTool (starting_position, 335, -386, 89 \Rx:=-1, \Ry:=18.3, \Rz:=0), v400, z1, Tooldata_7;
        MoveJ RelTool (starting_position, 333, -388, 87 \Rx:=-1.8, \Ry:=18, \Rz:=0), v400, z1, Tooldata_7;
        MoveJ RelTool (starting_position, 330, -390, 85 \Rx:=-2.6, \Ry:=18, \Rz:=0), v400, z1, Tooldata_7;
        MoveJ RelTool (starting_position, 327, -392, 83 \Rx:=-3.3, \Ry:=17.4, \Rz:=0), v400, z1, Tooldata_7;
        MoveJ RelTool (starting_position, 324, -394, 80 \Rx:=-3.9, \Ry:=16.8, \Rz:=0), v400, z1, Tooldata_7;
        MoveJ RelTool (starting_position, 321, -396, 78 \Rx:=-4.5, \Ry:=16.5, \Rz:=0), v400, z1, Tooldata_7;
        MoveJ RelTool (starting_position, 317, -398, 76 \Rx:=-5, \Ry:=15.9, \Rz:=0), v400, z1, Tooldata_7;
        MoveJ RelTool (starting_position, 313, -398, 73 \Rx:=-5.4, \Ry:=15.6, \Rz:=0), v400, z1, Tooldata_7;
        MoveJ RelTool (starting_position, 308, -400, 71 \Rx:=-5.7, \Ry:=15, \Rz:=0), v400, z1, Tooldata_7;
        MoveJ RelTool (starting_position, 304, -400, 69 \Rx:=-6, \Ry:=14.4, \Rz:=0), v400, z1, Tooldata_7;
        MoveJ RelTool (starting_position, 298, -400, 66 \Rx:=-6.2, \Ry:=13.5, \Rz:=0), v400, z1, Tooldata_7;
        MoveJ RelTool (starting_position, 293, -400, 64 \Rx:=-6.3, \Ry:=12.9, \Rz:=0), v400, z1, Tooldata_7;
        MoveJ RelTool (starting_position, 287, -400, 62 \Rx:=-6.3, \Ry:=12, \Rz:=0), v400, z1, Tooldata_7;
        MoveJ RelTool (starting_position, 281, -400, 59 \Rx:=-6.2, \Ry:=11.1, \Rz:=0), v400, z1, Tooldata_7;
        MoveJ RelTool (starting_position, 275, -400, 57 \Rx:=-5.9, \Ry:=10.2, \Rz:=0), v400, z1, Tooldata_7;
        MoveJ RelTool (starting_position, 268, -400, 56 \Rx:=-5.7, \Ry:=9.3, \Rz:=0), v400, z1, Tooldata_7;
        MoveJ RelTool (starting_position, 261, -400, 54 \Rx:=-5.4, \Ry:=8.4, \Rz:=0), v400, z1, Tooldata_7;
        MoveJ RelTool (starting_position, 254, -400, 52 \Rx:=-5.1, \Ry:=7.5, \Rz:=0), v400, z1, Tooldata_7;
        MoveJ RelTool (starting_position, 246, -400, 51 \Rx:=-4.6, \Ry:=6.3, \Rz:=0), v400, z1, Tooldata_7;
        MoveJ RelTool (starting_position, 239, -400, 49 \Rx:=-4.2, \Ry:=5.4, \Rz:=0), v400, z1, Tooldata_7;
        MoveJ RelTool (starting_position, 231, -400, 48 \Rx:=-3.6, \Ry:=4.2, \Rz:=0), v400, z1, Tooldata_7;
        MoveJ RelTool (starting_position, 224, -400, 48 \Rx:=-3.1, \Ry:=3.3, \Rz:=0), v400, z1, Tooldata_7;
        MoveJ RelTool (starting_position, 216, -400, 47 \Rx:=-2.6, \Ry:=2.1, \Rz:=0), v400, z1, Tooldata_7;
        MoveJ RelTool (starting_position, 208, -400, 46 \Rx:=-2, \Ry:=1.2, \Rz:=0), v400, z1, Tooldata_7;
        MoveJ RelTool (starting_position, 200, -400, 46 \Rx:=-1.3, \Ry:=0, \Rz:=0), v400, z1, Tooldata_7;
        MoveJ RelTool (starting_position, 192, -400, 46 \Rx:=-0.6, \Ry:=-1.2, \Rz:=0), v400, z1, Tooldata_7;
        MoveJ RelTool (starting_position, 185, -400, 46 \Rx:=0.2, \Ry:=-2.1, \Rz:=0), v400, z1, Tooldata_7;
        MoveJ RelTool (starting_position, 177, -400, 47 \Rx:=0.9, \Ry:=-3.3, \Rz:=0), v400, z1, Tooldata_7;
        MoveJ RelTool (starting_position, 170, -400, 47 \Rx:=1.7, \Ry:=-4.2, \Rz:=0), v400, z1, Tooldata_7;
        MoveJ RelTool (starting_position, 163, -400, 48 \Rx:=2.4, \Ry:=-5.4, \Rz:=0), v400, z1, Tooldata_7;
        MoveJ RelTool (starting_position, 156, -400, 49 \Rx:=3.1, \Ry:=-6.3, \Rz:=0), v400, z1, Tooldata_7;
        MoveJ RelTool (starting_position, 149, -400, 50 \Rx:=3.9, \Ry:=-7.2, \Rz:=0), v400, z1, Tooldata_7;
        MoveJ RelTool (starting_position, 143, -400, 52 \Rx:=4.5, \Ry:=-7.8, \Rz:=0), v400, z1, Tooldata_7;
        MoveJ RelTool (starting_position, 137, -400, 53 \Rx:=5.1, \Ry:=-8.7, \Rz:=0), v400, z1, Tooldata_7;
        MoveJ RelTool (starting_position, 131, -400, 55 \Rx:=5.7, \Ry:=-9.6, \Rz:=0), v400, z1, Tooldata_7;
        MoveJ RelTool (starting_position, 125, -400, 57 \Rx:=6.2, \Ry:=-10.2, \Rz:=0), v400, z1, Tooldata_7;
        MoveJ RelTool (starting_position, 120, -400, 59 \Rx:=6.6, \Ry:=-11.1, \Rz:=0), v400, z1, Tooldata_7;
        MoveJ RelTool (starting_position, 115, -400, 62 \Rx:=6.9, \Ry:=-11.7, \Rz:=0), v400, z1, Tooldata_7;
        MoveJ RelTool (starting_position, 110, -400, 64 \Rx:=7.2, \Ry:=-12.3, \Rz:=0), v400, z1, Tooldata_7;
        MoveJ RelTool (starting_position, 106, -400, 67 \Rx:=7.5, \Ry:=-12.9, \Rz:=0), v400, z1, Tooldata_7;
        MoveJ RelTool (starting_position, 102, -400, 69 \Rx:=7.6, \Ry:=-13.5, \Rz:=0), v400, z1, Tooldata_7;
        MoveJ RelTool (starting_position, 98, -400, 72 \Rx:=7.7, \Ry:=-14.1, \Rz:=0), v400, z1, Tooldata_7;
        MoveJ RelTool (starting_position, 95, -400, 74 \Rx:=7.6, \Ry:=-14.4, \Rz:=0), v400, z1, Tooldata_7;
        MoveJ RelTool (starting_position, 92, -400, 77 \Rx:=7.5, \Ry:=-15, \Rz:=0), v400, z1, Tooldata_7;
        MoveJ RelTool (starting_position, 89, -400, 79 \Rx:=7.3, \Ry:=-15.3, \Rz:=0), v400, z1, Tooldata_7;
        MoveJ RelTool (starting_position, 87, -400, 82 \Rx:=7, \Ry:=-15.6, \Rz:=0), v400, z1, Tooldata_7;
        MoveJ RelTool (starting_position, 85, -400, 84 \Rx:=6.6, \Ry:=-15.9, \Rz:=0), v400, z1, Tooldata_7;
        MoveJ RelTool (starting_position, 84, -400, 87 \Rx:=6.2, \Ry:=-15.9, \Rz:=0), v400, z1, Tooldata_7;
        MoveJ RelTool (starting_position, 82, -400, 89 \Rx:=5.7, \Ry:=-16.2, \Rz:=0), v400, z1, Tooldata_7;
        MoveJ RelTool (starting_position, 82, -400, 91 \Rx:=5.2, \Ry:=-16.2, \Rz:=0), v400, z1, Tooldata_7;
        MoveJ RelTool (starting_position, 81, -398, 94 \Rx:=4.6, \Ry:=-16.2, \Rz:=0), v400, z1, Tooldata_7;
        MoveJ RelTool (starting_position, 82, -398, 96 \Rx:=4, \Ry:=-16.2, \Rz:=0), v400, z1, Tooldata_7;
        MoveJ RelTool (starting_position, 82, -396, 98 \Rx:=3.3, \Ry:=-16.2, \Rz:=0), v400, z1, Tooldata_7;
        MoveJ RelTool (starting_position, 83, -394, 99 \Rx:=2.7, \Ry:=-15.9, \Rz:=0), v400, z1, Tooldata_7;
        MoveJ RelTool (starting_position, 83, -394, 101 \Rx:=2, \Ry:=-15.9, \Rz:=0), v400, z1, Tooldata_7;
        MoveJ RelTool (starting_position, 84, -392, 103 \Rx:=1.4, \Ry:=-15.6, \Rz:=0), v400, z1, Tooldata_7;
        MoveJ RelTool (starting_position, 86, -390, 104 \Rx:=0.8, \Ry:=-15.3, \Rz:=0), v400, z1, Tooldata_7;
        MoveJ RelTool (starting_position, 87, -388, 106 \Rx:=0.2, \Ry:=-15.3, \Rz:=0), v400, z1, Tooldata_7;
        MoveJ RelTool (starting_position, 88, -386, 107 \Rx:=-0.4, \Ry:=-15, \Rz:=0), v400, z1, Tooldata_7;
        MoveJ RelTool (starting_position, 89, -384, 108 \Rx:=-0.9, \Ry:=-14.7, \Rz:=0), v400, z1, Tooldata_7;
        MoveJ RelTool (starting_position, 90, -384, 109 \Rx:=-1.4, \Ry:=-14.4, \Rz:=0), v400, z1, Tooldata_7;
        MoveJ RelTool (starting_position, 91, -382, 110 \Rx:=-1.9, \Ry:=-14.1, \Rz:=0), v400, z1, Tooldata_7;
        MoveJ RelTool (starting_position, 92, -382, 111 \Rx:=-2.3, \Ry:=-13.8, \Rz:=0), v400, z1, Tooldata_7;






        !MoveJ [ [0, 0, 1225], [-0.282, 0.072, 0.956, 0.021], [0, -1,-1, 1], [0, 9E9, 9E9, 9E9, 9E9, 9E9] ],v20,z1,Tooldata_7;
        !MoveJ [ [0, 0, 1000], [-0.282, 0.072, 0.956, 0.021], [0, -1,-1, 1], [0, 9E9, 9E9, 9E9, 9E9, 9E9] ],v20,z1,Tooldata_7;
        !EGM_CARTESIAN_MOVE;
       ! RAPID_MOVE;

    ENDPROC

    ! ################################## Externally Guided motion (EGM) - Cartesian Control ################################## !



ENDMODULE
